FUNCTION A_UDINT : ST_Arg
VAR_INPUT
	nNumber	: REFERENCE TO UDINT;
END_VAR

IF __ISVALIDREF(nNumber) THEN
	A_UDINT.eType := E_ArgType.UDIntArg;
	A_UDINT.pData := ADR(nNumber);
	A_UDINT.nSize := SIZEOF(UDINT);
END_IF

END_FUNCTION

(* stored: Version 1.1.0.1, ProductVersion 3.1.4024.15
   POU A_UDINT: Id {a08428ad-331d-4af6-b92a-5f6242ccc9e1}, SpecialFunc None *)
